TYPE StepConfig :
STRUCT
	number		: INT;
	timeout		: TIME;
	
	description	: STRING;
END_STRUCT
END_TYPE

(* stored: Version 1.1.0.1, ProductVersion 3.1.4024.11
   DUT StepConfig: Id {b09cb353-48a0-4783-a699-dd3d03227ce5} *)
